FUNCTION TryConvert_STRING_TO_DATE : BOOL
VAR_INPUT
	in : STRING;
	out : REFERENCE TO DATE;
END_VAR

IF in <> DATE_TO_STRING(STRING_TO_DATE(in)) THEN
	RETURN;
END_IF

out := STRING_TO_DATE(in);
TryConvert_STRING_TO_DATE := TRUE;

END_FUNCTION

(* stored: Version 1.1.0.1, ProductVersion 3.1.4024.12
   POU TryConvert_STRING_TO_DATE: Id {70d162b9-ab5c-43ca-8f0a-71d691bfa891}, SpecialFunc None *)
